FUNCTION_BLOCK readTemp2
VAR
	fbRecGeneric		: 	FB_Rec_Generic;
END_VAR
VAR_INPUT
	sensorID			: DWORD;
END_VAR
VAR_OUTPUT
	tempOutput			: LREAL;
	humitityOut			: LREAL;
END_VAR

fbRecGeneric(str_KL6581 := GVL_EnOcean.stKL6581, byNode := 0, dw_ID := sensorID);

IF fbRecGeneric.bReceive = FALSE THEN
	tempOutput := F_Scale(fRawData := fbRecGeneric.ar_Value[1], fRawDataLowerOffLimit := 0, fRawDataUpperOffLimit := 255, fScaleDataLowerOffLimit := -20, fScaleDataUpperOffLimit := 60);
	humitityOut := F_Scale(fRawData := fbRecGeneric.ar_Value[2], fRawDataLowerOffLimit := 0, fRawDataUpperOffLimit := 255, fScaleDataLowerOffLimit := 0, fScaleDataUpperOffLimit := 100);
	
	Waardes.temp := tempOutput;
	Waardes.humitity := humitityOut;
	
END_IF

END_FUNCTION_BLOCK

(* stored: Version 1.1.0.1, ProductVersion 3.1.4024.2
   POU readTemp2: Id {17a03a96-4480-4b27-a861-f70573d50ab0}, SpecialFunc None *)
